{attribute 'linkalways'} 
{attribute 'no_explicit_call' := 'This FB is a CLASS and must be accessed using methods or properties'}
{attribute 'enable_dynamic_creation'}
FUNCTION_BLOCK FINAL AND_LINT EXTENDS Node
VAR
	in1 : _LINT(0);
	in2 : _LINT(0);
	out : _LINT(0);
END_VAR

METHOD PUBLIC Clone : I_Node
VAR
	pNode : POINTER TO AND_LINT;
END_VAR
pNode := __NEW(AND_LINT);
Clone := pNode^;
END_METHOD

METHOD FB_init : BOOL
VAR_INPUT
	bInitRetains : BOOL; // if TRUE, the retain variables are initialized (warm start / cold start)
	bInCopyCode : BOOL;  // if TRUE, the instance afterwards gets moved into the copy code (online change)
END_VAR
AddInput('in1',THIS^.in1);
AddInput('in2',THIS^.in2);
AddOutput('out', THIS^.out);
END_METHOD

METHOD PROTECTED OnExecute
VAR
END_VAR
out.Value := in1.Value AND in2.Value;
END_METHOD

END_FUNCTION_BLOCK

(* stored: Version 1.1.0.1, ProductVersion 3.1.4024.15
   POU AND_LINT: Id {83e6b195-422e-4b97-b98b-9ea29daadafd}, SpecialFunc None
   Folder Constructor: Id {b64bea68-100c-4554-ad2e-f15e090c3940}
   Method Clone: Id {6b3ca617-b0c5-43ec-bde2-94be7147f97d}
   Method FB_init: Id {5594fa9a-f489-4b3e-96a7-faafce0f461b}
   Method OnExecute: Id {29fd68b2-ec3e-4590-a7a2-780fffcb59b2} *)
